(*----------------------- Simple TCP/IP application. Adapt this code to match your needs. ----*)
FUNCTION_BLOCK FB_ServerApplication IMPLEMENTS I_Application
VAR
	_fbTx		: REFERENCE TO FB_FrameFifo;(* TX fifo *)
	_fbRx		: REFERENCE TO FB_FrameFifo;(* RX fifo *)
	_fbLog	 	: REFERENCE TO FB_LogFifo;(* Log/debug/error fifo *)
	_Updated : BOOL;
	
	sFromClient	: T_MaxString := '';
	sToClient	: T_MaxString := '';
	sLogMessage : T_MaxString := '';
	nCounter	: UDINT;
	nTempCounter : UDINT;
	
	ReceiveandSendData : I_Application;
END_VAR

PROPERTY fbLog : REFERENCE TO FB_LogFifo
GET
fbLog REF= _fbLog;
END_GET
SET
_fbLog REF= fbLog;
END_SET
END_PROPERTY

PROPERTY fbRx : REFERENCE TO FB_FrameFifo
GET
fbRx REF= _fbRx;
END_GET
SET
_fbRx REF= fbRx;
END_SET
END_PROPERTY

PROPERTY fbTx : REFERENCE TO FB_FrameFifo
GET
fbTx REF= _fbTx;
END_GET
SET
_fbTx REF= fbTx;
END_SET
END_PROPERTY

METHOD GetLogData
VAR_INPUT
END_VAR
fbLog.Remove( );
IF fbLog.bOk THEN
	
	(* TODO: Implement log message handler *)
	sLogMessage := fbLog.sGet;
END_IF
END_METHOD

{attribute 'monitoring':='call'}
PROPERTY isUpdated : BOOL
GET
isUpdated := _Updated;
END_GET
END_PROPERTY

METHOD Receive
fbRx.RemoveHead( );(* Fetch received string from rx fifo *)
	IF fbRx.bOk THEN(* Success *)

		(*TODO: Implement receive data handler *)
		nCounter := nCounter + 1;
		sFromClient := fbRx.sGet;
	END_IF

_Updated := SEL(nCounter = nTempCounter ,TRUE , FALSE);
nTempCounter := nCounter;
END_METHOD

METHOD Send
sToClient 	:= sFromClient;
(* Send received string back to the client *)
fbTx.AddTail( sPut := sToClient );(* Add string to the tx fifo *)
IF NOT fbTx.bOk THEN(* Fifo overflow => log error *)
	fbLog.Error( sMessage := 'FB_FrameFifo(sender)', nErrID := PLCPRJ_ERROR_SENDFIFO_OVERFLOW );
END_IF
END_METHOD

END_FUNCTION_BLOCK

(* stored: Version 1.1.0.1, ProductVersion 3.1.4024.12
   POU FB_ServerApplication: Id {fbb56189-ec16-45e6-9d9d-ffdcd266fc33}, SpecialFunc None
   Property fbLog: Id {94fe2199-a28d-4b10-89b6-7767c2e045dc}
   Get Get: Id {ca418fdb-0bc7-4915-bf0a-3ec1f444b54b}
   Set Set: Id {115ce44d-619f-4578-aa94-bc1354027357}
   Property fbRx: Id {ee77a888-8cde-41cb-a9f3-4f412a922755}
   Get Get: Id {9cb3754b-5c6f-40f4-b172-02aa28b753cc}
   Set Set: Id {179d8783-4b10-494c-be09-70246856946b}
   Property fbTx: Id {39d06f14-f109-437f-8570-8a18c683a51b}
   Get Get: Id {22b94075-8df1-45cf-af21-88b2e26f9c4e}
   Set Set: Id {dc755775-cc69-464a-b26f-2b2d59f55fb5}
   Method GetLogData: Id {2fca1445-3bd3-4cd4-be7c-f9e39800af7a}
   Property isUpdated: Id {d76cd531-efec-4a26-b4a0-939b55654e3b}
   Get Get: Id {2357f7eb-34c2-4d0a-8001-9933d8ca88c5}
   Method Receive: Id {64657dd0-0277-4642-bc82-19dcd1093786}
   Method Send: Id {862825d1-fbeb-405a-a22d-adc1535b753b} *)
